Fanuc TP program (LS listing): RECINIT.LS

/PROG  RECINIT
/ATTR
OWNER		= MNEDITOR;
COMMENT		= "RecInit";
PROG_SIZE	= 0;
CREATE		= DATE 26-01-01  TIME 00:00:00;
MODIFIED	= DATE 26-01-01  TIME 00:00:00;
FILE_NAME	= ;
VERSION		= 0;
LINE_COUNT	= 5;
MEMORY_SIZE	= 0;
PROTECT		= READ_WRITE;
TCD:  STACK_SIZE	= 0,
      TASK_PRIORITY	= 50,
      TIME_SLICE	= 0,
      BUSY_LAMP_OFF	= 0,
      ABORT_REQUEST	= 0,
      PAUSE_REQUEST	= 0;
DEFAULT_GROUP	= 1,*,*,*,*;
CONTROL_CODE	= 00000000 00000000;
/MN
   1:  !RAPID RecordProbe.RecInit ;
   2:  R[1:recCtrl.counter]=0    ;
   3:  !l.37 recCtrl.p.speed:=[400,500,5 ;
   4:  !l.38 recCtrl.p.zone:=z50 ;
   5:  F[1]=(OFF) ;
/POS
/END
